FUNCTION_BLOCK STRUCT_MUX (* Service Interface Function Block Type *)
  (* Standard: 61499-2; Description: Copyright (c) 2020 Johannes Kepler University Linz This program and the accompanying materials are made available under the terms of the Eclipse Public License 2.0 which is available at https://www.eclipse.org/legal/epl-2.0/ SPDX-License-Identifier: EPL-2.0 *)
  (* Version 3.0, 2025-04-14, Patrick Aigner, changed package *)
  PACKAGE eclipse4diac::convert;
  {SET_ATTRIBUTE(eclipse4diac::core::GenericClassName, 'GEN_STRUCT_MUX')}
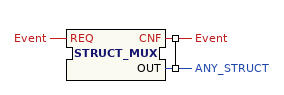
  EVENT_INPUT
    REQ; (* Normal Execution Request *)
  END_EVENT
  EVENT_OUTPUT
    CNF WITH OUT; (* Execution Confirmation *)
  END_EVENT
  VAR_OUTPUT
    OUT : ANY_STRUCT; (* Output *)
  END_VAR
END_FUNCTION_BLOCK
